// Mitsubishi GX Works2 project: 시퀀스 예제 1(경량화 시도)   PLC: Q03UDV

PROGRAM MAIN
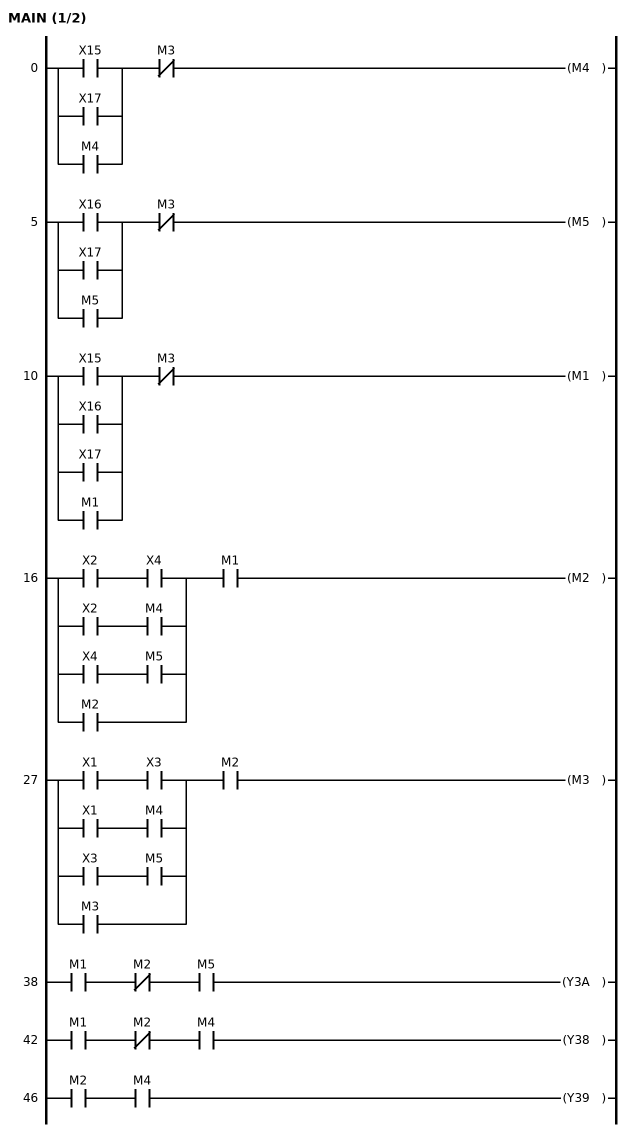
0     LD      X15
      OR      X17
      OR      M4
      ANI     M3
      OUT     M4
5     LD      X16
      OR      X17
      OR      M5
      ANI     M3
      OUT     M5
10    LD      X15
      OR      X16
      OR      X17
      OR      M1
      ANI     M3
      OUT     M1
16    LD      X2
      AND     X4
      LD      X2
      AND     M4
      ORB
      LD      X4
      AND     M5
      ORB
      OR      M2
      AND     M1
      OUT     M2
27    LD      X1
      AND     X3
      LD      X1
      AND     M4
      ORB
      LD      X3
      AND     M5
      ORB
      OR      M3
      AND     M2
      OUT     M3
38    LD      M1
      ANI     M2
      AND     M5
      OUT     Y3A
42    LD      M1
      ANI     M2
      AND     M4
      OUT     Y38
46    LD      M2
      AND     M4
      OUT     Y39
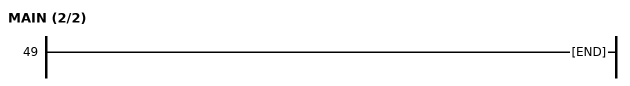
49    END
END_PROGRAM
